// TIA Portal V20 export
TYPE "LER_typeServoTorqueCalInterface"
// stored: Access Published
   STRUCT
      commands : "LER_typeServoTorqueCalCommands";
      monitoring : "LER_typeServoTorqueCalMonitoring";
      configuration : "LER_typeServoTorqueCalConfigruation";
   END_STRUCT;
END_TYPE
